TYPE ST_LogData:
  STRUCT
    bExecute: BOOL;
    sMsg    : STRING(MAX_STRING_LENGTH);
    sStation: STRING(20);
    nUserId : UDINT;
    eLogType: E_LogType;
  END_STRUCT
END_TYPE

(* stored: Version 1.1.0.1, ProductVersion 3.1.4024.2
   DUT ST_LogData: Id {293d680b-f29d-4b8c-ab2f-da3841baa15a} *)
